// TIA Portal V20 export
FUNCTION_BLOCK "LER_AlignVisionConversion"   // FB109, LAD
// stored: Access Published, MemoryReserve 100, SetENOAutomatically false
   VAR_INPUT
      VisionData : "LER_typeVisionMonitoring";
   END_VAR
   VAR_OUTPUT
      VisionDataConvert : "LER_typeVisionAlignResultData";
   END_VAR
BEGIN

REGION Network 1 (SCL)
   // Result
   #VisionDataConvert.tabFoldingMissingJudgementResult := 0.001 * DINT_TO_REAL(#VisionData.profinetInput.resultData248Byte_1.resultData[0]);
   #VisionDataConvert.electrodeLengthJudgementResult   := 0.001 * DINT_TO_REAL(#VisionData.profinetInput.resultData248Byte_1.resultData[1]);
   #VisionDataConvert.electrodeHeightJudgementResult   := 0.001 * DINT_TO_REAL(#VisionData.profinetInput.resultData248Byte_1.resultData[2]);

   // Measured value
   #VisionDataConvert.movementAmountAxisX1             := DINT_TO_REAL(#VisionData.profinetInput.resultData248Byte_1.resultData[3]);
   #VisionDataConvert.movementAmountAxisY1             := DINT_TO_REAL(#VisionData.profinetInput.resultData248Byte_1.resultData[4]);
   #VisionDataConvert.movementAmountAxisY2             := DINT_TO_REAL(#VisionData.profinetInput.resultData248Byte_1.resultData[5]);
   #VisionDataConvert.tabFoldingMissingReply           := DINT_TO_REAL(#VisionData.profinetInput.resultData248Byte_1.resultData[20]);
   #VisionDataConvert.tabFoldingMissingUpperRangeReply := DINT_TO_REAL(#VisionData.profinetInput.resultData248Byte_1.resultData[21]);
   #VisionDataConvert.tabFoldingMissingLowerRangeReply := DINT_TO_REAL(#VisionData.profinetInput.resultData248Byte_1.resultData[22]);
   #VisionDataConvert.electrodeLengthReply             := DINT_TO_REAL(#VisionData.profinetInput.resultData248Byte_1.resultData[23]);
   #VisionDataConvert.electrodeLengthUpperRangeReply   := DINT_TO_REAL(#VisionData.profinetInput.resultData248Byte_1.resultData[24]);
   #VisionDataConvert.electrodeLengthLowerRangeReply   := DINT_TO_REAL(#VisionData.profinetInput.resultData248Byte_1.resultData[25]);
   #VisionDataConvert.electrodeHeightReply             := DINT_TO_REAL(#VisionData.profinetInput.resultData248Byte_1.resultData[26]);
   #VisionDataConvert.electrodeHeightUpperRangeReply   := DINT_TO_REAL(#VisionData.profinetInput.resultData248Byte_1.resultData[27]);
   #VisionDataConvert.electrodeHeightLowerRangeReply   := DINT_TO_REAL(#VisionData.profinetInput.resultData248Byte_1.resultData[28]);
END_REGION
END_FUNCTION_BLOCK
